FUNCTION_BLOCK MILLING_APPROACH_DATA_MANAGER (* Approach strategy manager *)
  (* Standard: 61499-2 *)
  (* Version 1.0, 17-05-12, GASR, Universidade do Estado de Santa Catarina *)
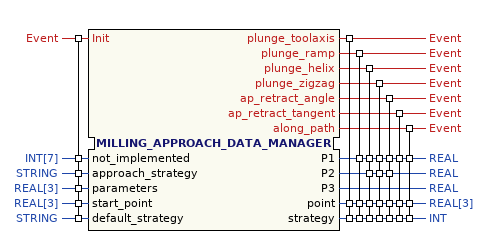
  EVENT_INPUT
    Init WITH not_implemented, approach_strategy, parameters, start_point, default_strategy;
  END_EVENT
  EVENT_OUTPUT
    plunge_toolaxis WITH point, strategy;
    plunge_ramp WITH point, strategy, P1;
    plunge_helix WITH point, strategy, P1, P2;
    plunge_zigzag WITH point, strategy, P1, P2;
    ap_retract_angle WITH point, strategy, P1, P2;
    ap_retract_tangent WITH point, strategy, P1;
    along_path WITH point, strategy, P1;
  END_EVENT
  VAR_INPUT
    not_implemented : ARRAY [0..6] OF INT; (* list of not implemented strategies *)
    approach_strategy : STRING;
    parameters : ARRAY [0..2] OF REAL;
    start_point : ARRAY [0..2] OF REAL;
    default_strategy : STRING := 'plunge_tool_axis';
  END_VAR
  VAR_OUTPUT
    P1 : REAL;
    P2 : REAL;
    P3 : REAL;
    point : ARRAY [0..2] OF REAL;
    strategy : INT;
  END_VAR
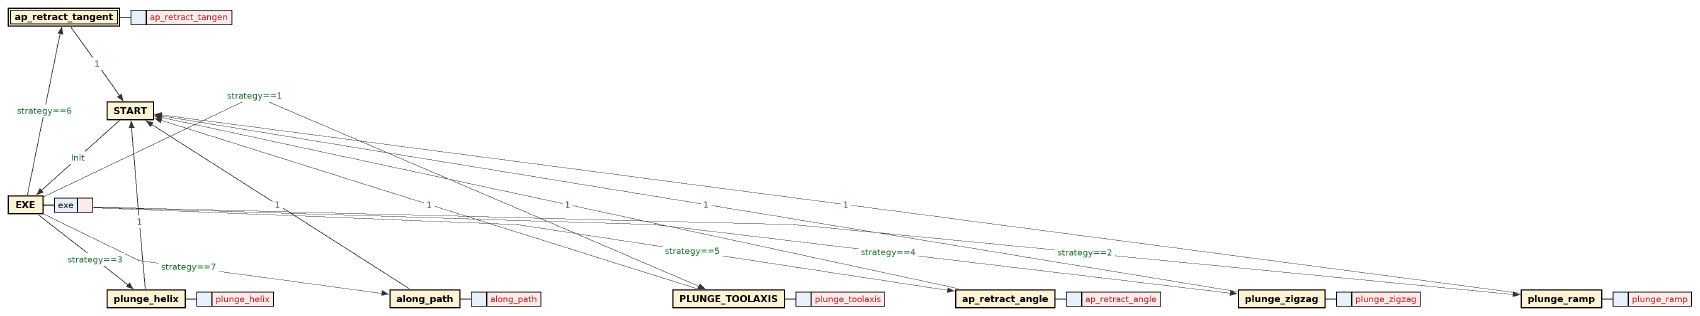
  EC_STATES
    ap_retract_tangent : -> ap_retract_tangen;
    plunge_helix : -> plunge_helix;
    along_path : -> along_path;
    EXE : exe;
    PLUNGE_TOOLAXIS : -> plunge_toolaxis;
    ap_retract_angle : -> ap_retract_angle;
    START;
    plunge_zigzag : -> plunge_zigzag;
    plunge_ramp : -> plunge_ramp;
  END_STATES
  EC_TRANSITIONS
    ap_retract_tangent TO START := 1;
    plunge_helix TO START := 1;
    along_path TO START := 1;
    EXE TO PLUNGE_TOOLAXIS := strategy==1;
    EXE TO plunge_ramp := strategy==2;
    EXE TO plunge_helix := strategy==3;
    EXE TO plunge_zigzag := strategy==4;
    EXE TO ap_retract_angle := strategy==5;
    EXE TO ap_retract_tangent := strategy==6;
    EXE TO along_path := strategy==7;
    PLUNGE_TOOLAXIS TO START := 1;
    ap_retract_angle TO START := 1;
    START TO EXE := Init;
    plunge_zigzag TO START := 1;
    plunge_ramp TO START := 1;
  END_TRANSITIONS
  ALGORITHM exe IN Lua:
local id = {
PLUNGE_TOOLAXIS    = 1,
PLUNGE_RAMP        = 2,
PLUNGE_HELIX       = 3,
PLUNGE_ZIGZAG      = 4,
AP_RETRACT_ANGLE   = 5,
AP_RETRACT_TANGENT = 6,
ALONG_PATH         = 7,
}
strategy = id[ approach_strategy ]
for k,v in pairs( not_implemented ) do
    if( strategy == v ) then
        strategy = 1
        break
    end
end
point[1] = start_point[1]
point[2] = start_point[2]
point[3] = start_point[3]
  END_ALGORITHM
END_FUNCTION_BLOCK
